FUNCTION_BLOCK FB_Axis
VAR_INPUT
	//axis		:AXIS_REF;
	
END_VAR
VAR_OUTPUT
END_VAR
VAR	
	fbPower: MC_Power;
END_VAR

METHOD PowerOn : BOOL
VAR_INPUT
END_VAR
fbPower(
	Axis:=GVL_General.Axis1 , 
	Enable:= GVL_General.bPowerOn,
	Enable_Positive:=TRUE , 
	Enable_Negative:= TRUE, 
	Override:= , 
	BufferMode:= , 
	Options:= ,
	Status=> , 
	Busy=> , 
	Active=> , 
	Error=> , 
	ErrorID=> );
END_METHOD

END_FUNCTION_BLOCK

(* stored: Version 1.1.0.1, ProductVersion 3.1.4022.16
   POU FB_Axis: Id {a59f5d40-768d-47ee-b53a-dd3069670267}, SpecialFunc None
   Method PowerOn: Id {92beff14-75f0-4a0e-843e-31ea1c1ea9ee} *)
